// TIA Portal V20 export
DATA_BLOCK "SafetyDoorInterface"   // DB188
// stored: MemoryReserve 100
   VAR
      "FDoorEC.LH" { ExternalWritable := 'False'} : "LER_typefDoorInterface";
      "FDoorEC.RH" { ExternalWritable := 'False'} : "LER_typefDoorInterface";
      "FDoorEC.Top" { ExternalWritable := 'False'} : "LER_typefDoorInterface";
      FDoorCutter : "LER_typefDoorInterface";
      FDoorMagazine : "LER_typefDoorInterface";
      FDoorConveyor : "LER_typefDoorInterface";
      FDoorCentralAisle : "LER_typefDoorInterface";
   END_VAR
BEGIN
   "FDoorEC.LH".configuration.referenceDesignator := WSTRING#'LH';
   "FDoorEC.RH".configuration.referenceDesignator := WSTRING#'RH';
   "FDoorEC.Top".configuration.referenceDesignator := WSTRING#'Main';
   FDoorCutter.configuration.referenceDesignator := WSTRING#'Cutter';
   FDoorMagazine.configuration.referenceDesignator := WSTRING#'Magazine';
   FDoorConveyor.configuration.referenceDesignator := WSTRING#'C/V';
   FDoorCentralAisle.configuration.referenceDesignator := WSTRING#'Central';
END_DATA_BLOCK
